(* PLC project SafeLOGIC, BrAutomation SafeDESIGNER  5.24.1.0 *)
(* stored: companyURL http://www.br-automation.com, creationDateTime Mon Dec 15 17:53:00 2025 *)

PROGRAM Main

(* FBD diagram, written out as Structured Text *)
(* Function 05/06 - Engine cooling water pressure min/maximum *)
(* Actual ECW pressure before pump [mbar] *)
xSCALE_F05_AI_Pr_ECW(sX := sAI_Pr_ECW, sX1 := SAFEDINT#4000, sX2 := SAFEDINT#20000, sY1 := SAFEDINT#0, sY2 := SAFEDINT#10000, sbSafeCurrentOK := sbSafeCurrentOK_AI_Pr_ECW);
siPr_ECW := xSCALE_F05_AI_Pr_ECW.sY_Scal;
(* Alarm *)
(* Safety loop *)
bAMM_A2397 := xSCALE_F05_AI_Pr_ECW.bAMM_MSF;
iOUT_F05_Pr_ECW := xSCALE_F05_AI_Pr_ECW.iOUT_Y_Scal;
(* Measurement signal OK *)
sbPr_ECW_MsOK := xSCALE_F05_AI_Pr_ECW.sbMsOK;
sbSL_OK_ECW_Ms := xSCALE_F05_AI_Pr_ECW.sbSL_OK;
(* Actual ECW pressure after pump [mbar] *)
xSCALE_F06_AI_Pr_ECWaP(sX := sAI_Pr_ECWaP, sX1 := SAFEDINT#4000, sX2 := SAFEDINT#20000, sY1 := SAFEDINT#0, sY2 := SAFEDINT#10000, sbSafeCurrentOK := sbSafeCurrentOK_AI_Pr_ECWaP);
siPr_ECWaP := xSCALE_F06_AI_Pr_ECWaP.sY_Scal;
(* Alarm *)
(* Safety loop *)
bAMM_A9411 := xSCALE_F06_AI_Pr_ECWaP.bAMM_MSF;
iOUT_F06_Pr_ECWaP := xSCALE_F06_AI_Pr_ECWaP.iOUT_Y_Scal;
(* Measurement signal OK *)
sbPr_ECWaP_MsOK := xSCALE_F06_AI_Pr_ECWaP.sbMsOK;
sbSL_OK_ECWaP_Ms := xSCALE_F06_AI_Pr_ECWaP.sbSL_OK;
(* Check ECW Pumps off *)
(* All ECW pumps off for 2min *)
(* Elapsed time *)
xELAPSED_TIME_ECW(IN := BOOL_TO_SAFEBOOL(bIN_ECW_PumpsOff), PT := SAFETIME#120s);
sbECW_PumpsOff_120s := xELAPSED_TIME_ECW.Q;
iOUT_F06_ECW_PumpsOff_2m_ET := xELAPSED_TIME_ECW.iOUT_ET;
(* Pressure Minimum *)
(* Alarm *)
xKeepAMM_2s_A2396(sbAMMxxxx := OR_S(GE_S(siPr_ECW, PARA_Pr_ECW_LoLo), sbGasValves_Closed, NOT_S(sbPr_ECW_MsOK)));
bAMM_A2396 := xKeepAMM_2s_A2396.bAMMxxxx;
(* Pressure difference calculation *)
(* Pressure difference [mbar] *)
xDEV_ECW(sInput_1 := siPr_ECWaP, sInput_2 := siPr_ECW);
iOUT_F05_Pr_ECW_Diff := xDEV_ECW.iOUT_Diff;
(* Pressure difference OK *)
sbPr_ECW_DiffOK := xDEV_ECW.sbDiffOK;
siPr_ECW_Diff := xDEV_ECW.sDiff;
bOUT_F05_Pr_ECW_DiffOK := xDEV_ECW.bOUT_DiffOK;
(* AT STILLSTAND: Maximum deviation to pressure sensor after pump *)
(* Alarm *)
xKeepAMM_2s_A2398(sbAMMxxxx := NOT_S(AND_S(OR_S(GT_S(siPr_ECW_Diff, PARA_Pr_ECW_HiHi_Diff), NOT_S(sbPr_ECW_DiffOK)), sbN_Standstill, sbECW_PumpsOff_120s, sbPr_ECW_MsOK, sbPr_ECWaP_MsOK)));
bAMM_A2398 := xKeepAMM_2s_A2398.bAMMxxxx;
(* Difference pressure minimum *)
(* Alarm *)
xTON_F06_Nom90(IN := sbN_EngAct_Nom90, PT := SAFETIME#120s);
xTOF_F06_DPr(IN := NOT_S(AND_S(OR_S(LT_S(siPr_ECW_Diff, PARA_DPr_ECWP_LoLo), NOT_S(sbPr_ECW_DiffOK)), sbPr_ECW_MsOK, sbPr_ECWaP_MsOK, OR_S(sbGCB_On_10s, xTON_F06_Nom90.Q))), PT := SAFETIME#10s);
xKeepAMM_2s_A9434(sbAMMxxxx := xTOF_F06_DPr.Q);
bAMM_A9434 := xKeepAMM_2s_A9434.bAMMxxxx;
(* Pressure Maximum (Sensor drift) *)
(* Alarm *)
xTOF_F05_Pr_ECW_HiHi(IN := LE_S(siPr_ECW, PARA_Pr_ECW_HiHi_Check), PT := SAFETIME#10s);
xKeepAMM_2s_A9408(sbAMMxxxx := OR_S(xTOF_F05_Pr_ECW_HiHi.Q, NOT_S(sbPr_ECW_MsOK)));
bAMM_A9408 := xKeepAMM_2s_A9408.bAMMxxxx;
(* Frozen sensor value *)
(* Alarm *)
(* Elapsed time *)
xFROZEN_ECW(siPr := siPr_ECW, siPr_saved := siPr_ECW_Saved, sbGV_Closed := sbGasValves_Closed, sbN_Nom90_10s := sbN_EngAct_Nom90_10s);
iOUT_F05_Pr_ECW_Fr_1m_ET := xFROZEN_ECW.iOUT_Pr_Frozen_1m_ET;
bAMM_A9409 := xFROZEN_ECW.bError_Frozen;
(* Save actual value *)
siPr_ECW_Saved := siPr_ECW;
(* Safety loop *)
(* Safety loop *)
sbF05_OK_ECW_Pr_Min := AND_S(BOOL_TO_SAFEBOOL(bAMM_A2396), sbSL_OK_ECW_Ms, BOOL_TO_SAFEBOOL(bAMM_A2398), BOOL_TO_SAFEBOOL(bAMM_A9408), BOOL_TO_SAFEBOOL(bAMM_A9409));
(* HMI - ECW pressure min OK *)
(* ECW pressure MIN OK *)
bOUT_F05_OK := SAFEBOOL_TO_BOOL(AND_S(sbN_EngAct_Nom90_10s, sbGasValves_Open, sbF05_OK_ECW_Pr_Min));
(* Release signal after error *)
(* Reset channel error *)
sbSafeRelease_AI_Pr_ECW := BOOL_TO_SAFEBOOL(bIN_Reset_sPLC);
(* Pressure Maximum *)
(* Alarm *)
xKeepAMM_2s_A9410(sbAMMxxxx := OR_S(LT_S(siPr_ECWaP, PARA_Pr_ECWaP_HiHi), NOT_S(sbPr_ECWaP_MsOK)));
bAMM_A9410 := xKeepAMM_2s_A9410.bAMMxxxx;
(* Frozen sensor value *)
(* Alarm *)
(* Elapsed time *)
xFROZEN_ECWaP(siPr := siPr_ECWaP, siPr_saved := siPr_ECWaP_Saved, sbGV_Closed := sbGasValves_Closed, sbN_Nom90_10s := sbN_EngAct_Nom90_10s);
iOUT_F06_Pr_ECWaP_Fr_1m_ET := xFROZEN_ECWaP.iOUT_Pr_Frozen_1m_ET;
bAMM_A9412 := xFROZEN_ECWaP.bError_Frozen;
(* Save actual value *)
siPr_ECWaP_Saved := siPr_ECWaP;
(* Safety loop *)
(* Safety loop *)
sbF06_OK_ECW_Pr_Max := AND_S(BOOL_TO_SAFEBOOL(bAMM_A9410), sbSL_OK_ECWaP_Ms, BOOL_TO_SAFEBOOL(bAMM_A9412), BOOL_TO_SAFEBOOL(bAMM_A9434));
(* HMI - ECW pressure max OK *)
(* ECW pressure MAX OK *)
bOUT_F06_OK := SAFEBOOL_TO_BOOL(AND_S(sbN_EngAct_Nom90_10s, sbGasValves_Open, sbF06_OK_ECW_Pr_Max));
(* Release signal after error *)
(* Reset channel error *)
sbSafeRelease_AI_Pr_ECWaP := BOOL_TO_SAFEBOOL(bIN_Reset_sPLC);
END_PROGRAM
